(* PLC project CodesysTest.project, PN2IC PLCopen CODESYS V3.5 SP17 Patch 3 *)
(* stored: creationDateTime 2022-12-17T23:12:03, modificationDateTime 2022-12-17T23:12:03 *)

PROGRAM flow_teste

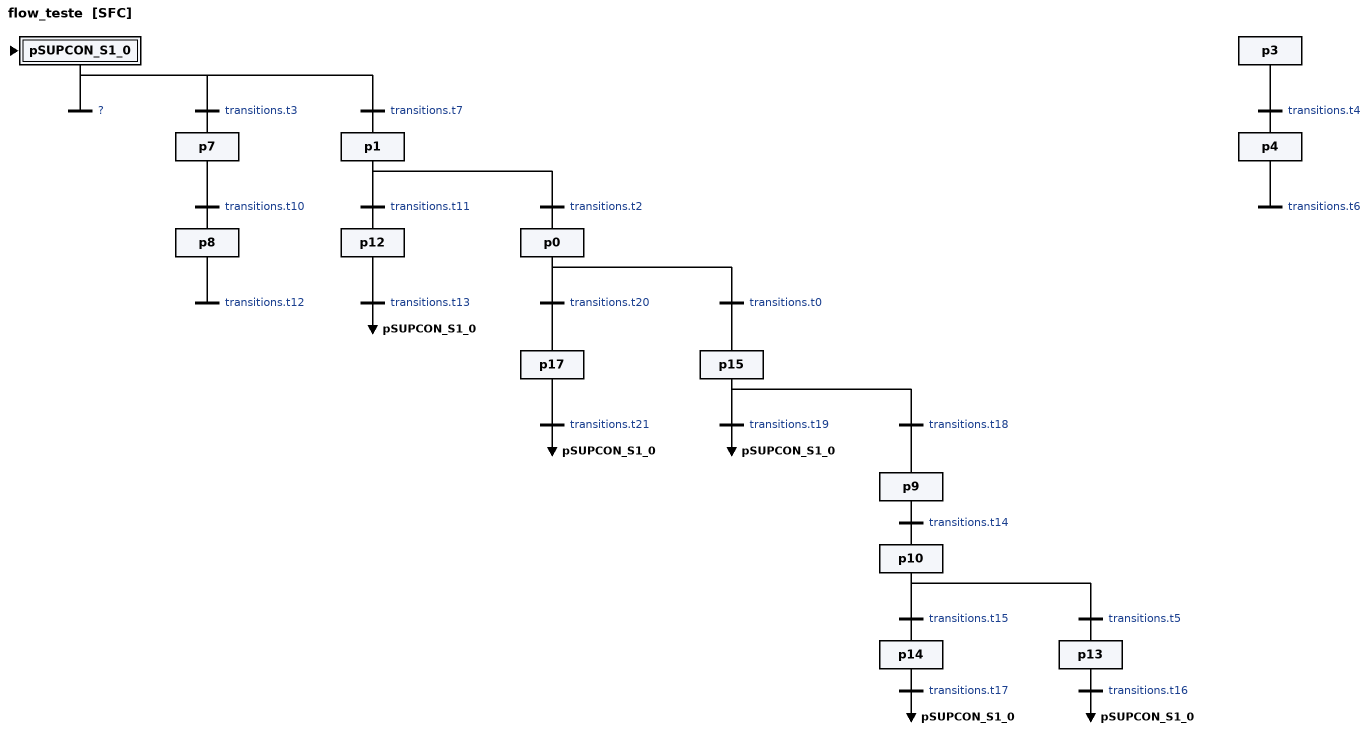
INITIAL_STEP pSUPCON_S1_0:
END_STEP
TRANSITION FROM pSUPCON_S1_0 TO ?
  := ?;
END_TRANSITION
TRANSITION FROM pSUPCON_S1_0 TO p7
  := transitions.t3;
END_TRANSITION
TRANSITION FROM pSUPCON_S1_0 TO p1
  := transitions.t7;
END_TRANSITION
STEP p3:
END_STEP
TRANSITION FROM p3 TO p4
  := transitions.t4;
END_TRANSITION
STEP p4:
END_STEP
TRANSITION FROM p4 TO ?
  := transitions.t6;
END_TRANSITION
STEP p7:
END_STEP
TRANSITION FROM p7 TO p8
  := transitions.t10;
END_TRANSITION
STEP p8:
END_STEP
TRANSITION FROM p8 TO ?
  := transitions.t12;
END_TRANSITION
STEP p1:
END_STEP
TRANSITION FROM p1 TO p12
  := transitions.t11;
END_TRANSITION
TRANSITION FROM p1 TO p0
  := transitions.t2;
END_TRANSITION
STEP p12:
END_STEP
TRANSITION FROM p12 TO pSUPCON_S1_0
  := transitions.t13;
END_TRANSITION
STEP p0:
END_STEP
TRANSITION FROM p0 TO p17
  := transitions.t20;
END_TRANSITION
TRANSITION FROM p0 TO p15
  := transitions.t0;
END_TRANSITION
STEP p17:
END_STEP
TRANSITION FROM p17 TO pSUPCON_S1_0
  := transitions.t21;
END_TRANSITION
STEP p15:
END_STEP
TRANSITION FROM p15 TO pSUPCON_S1_0
  := transitions.t19;
END_TRANSITION
TRANSITION FROM p15 TO p9
  := transitions.t18;
END_TRANSITION
STEP p9:
END_STEP
TRANSITION FROM p9 TO p10
  := transitions.t14;
END_TRANSITION
STEP p10:
END_STEP
TRANSITION FROM p10 TO p14
  := transitions.t15;
END_TRANSITION
TRANSITION FROM p10 TO p13
  := transitions.t5;
END_TRANSITION
STEP p14:
END_STEP
TRANSITION FROM p14 TO pSUPCON_S1_0
  := transitions.t17;
END_TRANSITION
STEP p13:
END_STEP
TRANSITION FROM p13 TO pSUPCON_S1_0
  := transitions.t16;
END_TRANSITION
END_PROGRAM

PROGRAM transitions

         
        
END_PROGRAM

CONFIGURATION Application
  RESOURCE Application ON PLC
    VAR_GLOBAL  (* GVL *)
      t10 : BOOL;
      t11 : BOOL;
      t12 : BOOL;
      t13 : BOOL;
      t14 : BOOL;
      t15 : BOOL;
      t16 : BOOL;
      t17 : BOOL;
      t18 : BOOL;
      t19 : BOOL;
      t2 : BOOL;
      t20 : BOOL;
      t21 : BOOL;
      t3 : BOOL;
      t4 : BOOL;
      t5 : BOOL;
      t6 : BOOL;
      t7 : BOOL;
      t0 : BOOL;
      t1 : BOOL;
    END_VAR
    TASK MainTask(INTERVAL := T#20ms, PRIORITY := 1);
    PROGRAM flow_teste WITH MainTask : flow_teste;
  END_RESOURCE
END_CONFIGURATION
